(* CODESYS project string-builder-unit-test-history

Project tree, tasks and I/O mapping:
  Device : CODESYS Control Win V3 x64, 3S - Smart Software Solutions GmbH, version 3.5.17.20
    application Application
      libraries: Standard, 3.5.18.0 (System); co♻e - A unittest framework for CODESYS, 1.2.0.0 (www.co5e.org); StringBuilder, 0.0.0.1 (PowerCore Engineering)
      task MainTask (cyclic, interval t#20ms, priority 1) calls PLC_PRG
      function block FB_TestSuite_withBuffer [ST]: AssertEquals_Buffer
      FunctionBlocks/
        function block UT_StringBuilder [ST]: T001_Append, T002_Reset
        function block UT_StringBuilderExt [ST]: T001_Append, T002_Reset
      Functions/
        function block UT_ANY_TO_HEXSTR [ST]: T001_Test
        function block UT_ANY_TO_NUMSTRING [ST]: T001_Test
        function block UT_FindFormat [ST]: T001_FindFormat
        function block UT_Format_1 [ST]: T001_Format_1
        function block UT_Format [ST]: T001_Format_2, T002_Format_3, T003_Format_4, T004_Format_5, T005_Format_6, T006_Format_7, T007_Format_8, T008_Format_9, T009_Format_10, T010_Format_2
        function block UT_FormatExt_1 [ST]: T001_Format_1
        function block UT_FormatExt [ST]: T001_FormatExt_2, T002_FormatExt_3, T003_FormatExt_4, T004_FormatExt_5, T005_FormatExt_6, T006_FormatExt_7, T007_FormatExt_8, T008_FormatExt_9, T009_FormatExt_10, T010_FormatExt_2
      program PLC_PRG [ST]
*)

// Device/Application/PLC_PRG
PROGRAM PLC_PRG
VAR
	utStringBuilder : UT_StringBuilder;
	utFindFormat : UT_FindFormat;
	utFormat_1 : UT_Format_1;
	utFormat : UT_Format;
END_VAR

coUnit.RUN();

END_PROGRAM

// Device/Application/FunctionBlocks/UT_StringBuilder
FUNCTION_BLOCK UT_StringBuilder EXTENDS coUnit.FB_TestSuite
VAR_INPUT
END_VAR
VAR_OUTPUT
END_VAR
VAR
END_VAR

T001_Append();
T002_Reset();

METHOD T001_Append
VAR_INPUT
END_VAR
VAR
	sb : PSB.StringBuilder;
END_VAR
TEST('T001_Append');

sb.Append('Hello');
sb.Append(', ');
sb.Append('world!');

AssertEquals_STRING('Hello, world!', sb.sOutput, 'Unexpected result');

TEST_FINISHED();
END_METHOD

METHOD T002_Reset
VAR_INPUT
END_VAR
VAR
	sb : PSB.StringBuilder;
END_VAR
TEST('T002_Reset');

sb.Append('Hello, world!');

AssertEquals_STRING('Hello, world!', sb.sOutput, 'Unexpected result');

sb.Reset();
AssertEquals_STRING('', sb.sOutput, 'Unexpected result');

TEST_FINISHED();
END_METHOD

END_FUNCTION_BLOCK

// Device/Application/Functions/UT_FindFormat
FUNCTION_BLOCK UT_FindFormat EXTENDS coUnit.FB_TestSuite
VAR_INPUT
END_VAR
VAR_OUTPUT
END_VAR
VAR
END_VAR

T001_FindFormat('This {} thing', start:=0, sl_start:=6, sl_end:=7);
T001_FindFormat('{} thing', start:=0, sl_start:=1, sl_end:=2);
T001_FindFormat('thing', start:=0, sl_start:=0, sl_end:=0);
T001_FindFormat('This {} thing {}', start:=7, sl_start:=15, sl_end:=16);

METHOD T001_FindFormat
VAR_INPUT
	sFmtStr : STRING(255);
	start : DINT;
	sl_start : DINT;
	sl_end : DINT;
END_VAR
VAR
	slResult : PSB.slice;
END_VAR
TEST(concat(concat('T001_FindFormat:', sFmtStr), concat(concat('-', DINT_TO_STRING(start)), 
	concat(concat('-' , TO_STRING(sl_start)), concat('-', TO_STRING(sl_end)))))); 

slResult := PSB.FindFormat(sFmtStr, start);

AssertEquals_DINT(sl_start, slResult.start, 'Unexpected start position');
AssertEquals_DINT(sl_end, slResult.end, 'Unexpected end position');

TEST_FINISHED();
END_METHOD

END_FUNCTION_BLOCK

// Device/Application/Functions/UT_Format_1
FUNCTION_BLOCK UT_Format_1 EXTENDS coUnit.FB_TestSuite
VAR_INPUT
END_VAR
VAR_OUTPUT
END_VAR
VAR
END_VAR

T001_Format_1('Hello, {}!', 'world', 'Hello, world!');
T001_Format_1('Hello {}', 'john', 'Hello john');

METHOD T001_Format_1
VAR_INPUT
	fmtstr : STRING(255);
	str1 : STRING(255);
	sExpected : STRING(255);
END_VAR
VAR
	sResult : STRING(255);
END_VAR
TEST(concat(concat('T001_Format_1:', fmtstr), concat('-', str1)));

sResult := PSB.Format_1(fmtstr, str1);

AssertEquals_STRING(sExpected, sResult, 'unexpected result');

TEST_FINISHED();
END_METHOD

END_FUNCTION_BLOCK

// Device/Application/Functions/UT_Format
FUNCTION_BLOCK UT_Format EXTENDS coUnit.FB_TestSuite
VAR_INPUT
END_VAR
VAR_OUTPUT
END_VAR
VAR
END_VAR

T001_Format_2('Hello, {}! Goodbye {} world.',
              'world',
              'cruel',
              'Hello, world! Goodbye cruel world.');
T002_Format_3('{}-{}-{}',
	'a',
	'b',
	'c',
	'a-b-c');
T003_Format_4('{}-{}-{}-{}-',
	'1',
	'2',
	'3',
	'4',
	'1-2-3-4-');
// missing format element
T004_Format_5('{}-{}-{}-{}-',
	'1',
	'2',
	'3',
	'4',
	'5',
	'1-2-3-4-');
	
// extra format element
T004_Format_5('{}-{}-{}-{}-{}-{}',
	'1',
	'2',
	'3',
	'4',
	'5',
	'1-2-3-4-5-{}');
T005_Format_6('{}-{}-{}-{}-{}-{}',
	INT_TO_STRING(1),
	TO_STRING(123.456),
	'c',
	'd',
	'e',
	'f',
	'1-123.456-c-d-e-f');
T006_Format_7('{}-{}-{}-{}-{}-{}-{}',
	'1', '2', '3', '4', '5', '6', '7',
	'1-2-3-4-5-6-7');
T007_Format_8('{}-{}-{}-{}-{}-{}-{}-{}',
	'1', '2', '3', '4', '5', '6', '7','8',
	'1-2-3-4-5-6-7-8');
T008_Format_9('{}-{}-{}-{}-{}-{}-{}-{}-{}',
	'1', '2', '3', '4', '5', '6', '7','8','9',
	'1-2-3-4-5-6-7-8-9');
T009_Format_10('{}-{}-{}-{}-{}-{}-{}-{}-{}-{}',
	'1', '2', '3', '4', '5', '6', '7','8','9','10',
	'1-2-3-4-5-6-7-8-9-10');
T010_Format_2('test-with-to-string-input-int:{}-real:{}', 123, 456.789, 'test-with-to-string-input-int:123-real:456.789');

METHOD T001_Format_2
VAR_INPUT
	fmtstr : STRING(255);
	str1 : STRING(255);
	str2 : STRING(255);
	sExpected : STRING(255);
END_VAR
VAR_INST
	sResult : STRING(255);
END_VAR
TEST(concat(concat('T001_Format_2:', fmtstr), concat('-', sExpected)));

sResult := PSB.Format_2(fmtstr, str1, str2);

AssertEquals_STRING(sExpected, sResult, 'unexpected result');

TEST_FINISHED();
END_METHOD

METHOD T002_Format_3
VAR_INPUT
	fmtstr : STRING(255);
	str1 : STRING(255);
	str2 : STRING(255);
	str3 : STRING(255);
	sExpected : STRING(255);
END_VAR
VAR_INST
	sResult : STRING(255);
END_VAR
TEST(concat(concat('T001_Format_3:', fmtstr), concat('-', sExpected)));

sResult := PSB.Format_3(fmtstr, str1, str2, str3);

AssertEquals_STRING(sExpected, sResult, 'unexpected result');

TEST_FINISHED();
END_METHOD

METHOD T003_Format_4
VAR_INPUT
	fmtstr : STRING(255);
	str1 : STRING(255);
	str2 : STRING(255);
	str3 : STRING(255);
	str4 : STRING(255);
	sExpected : STRING(255);
END_VAR
VAR_INST
	sResult : STRING(255);
END_VAR
TEST(concat(concat('T003_Format_4:', fmtstr), concat('-', sExpected)));

sResult := PSB.Format_4(fmtstr, str1, str2, str3, str4);

AssertEquals_STRING(sExpected, sResult, 'unexpected result');

TEST_FINISHED();
END_METHOD

METHOD T004_Format_5
VAR_INPUT
	fmtstr : STRING(255);
	str1 : STRING(255);
	str2 : STRING(255);
	str3 : STRING(255);
	str4 : STRING(255);
	str5 : STRING(255);
	sExpected : STRING(255);
END_VAR
VAR_INST
	sResult : STRING(255);
END_VAR
TEST(concat(concat('T004_Format_5:', fmtstr), concat('-', sExpected)));

sResult := PSB.Format_5(fmtstr, str1, str2, str3, str4, str5);

AssertEquals_STRING(sExpected, sResult, 'unexpected result');

TEST_FINISHED();
END_METHOD

METHOD T005_Format_6
VAR_INPUT
	fmtstr : STRING(255);
	str1 : STRING(255);
	str2 : STRING(255);
	str3 : STRING(255);
	str4 : STRING(255);
	str5 : STRING(255);
	str6 : STRING(255);
	sExpected : STRING(255);
END_VAR
VAR_INST
	sResult : STRING(255);
END_VAR
TEST(concat(concat('T005_Format_6:', fmtstr), concat('-', sExpected)));

sResult := PSB.Format_6(fmtstr, str1, str2, str3, str4, str5, str6);

AssertEquals_STRING(sExpected, sResult, 'unexpected result');

TEST_FINISHED();
END_METHOD

METHOD T006_Format_7
VAR_INPUT
	fmtstr : STRING(255);
	str1 : STRING(255);
	str2 : STRING(255);
	str3 : STRING(255);
	str4 : STRING(255);
	str5 : STRING(255);
	str6 : STRING(255);
	str7 : STRING(255);
	sExpected : STRING(255);
END_VAR
VAR_INST
	sResult : STRING(255);
END_VAR
TEST(concat(concat('T006_Format_7:', fmtstr), concat('-', sExpected)));

sResult := PSB.Format_7(fmtstr, str1, str2, str3, str4, str5, str6, str7);

AssertEquals_STRING(sExpected, sResult, 'unexpected result');

TEST_FINISHED();
END_METHOD

METHOD T007_Format_8
VAR_INPUT
	fmtstr : STRING(255);
	str1 : STRING(255);
	str2 : STRING(255);
	str3 : STRING(255);
	str4 : STRING(255);
	str5 : STRING(255);
	str6 : STRING(255);
	str7 : STRING(255);
	str8 : STRING(255);
	sExpected : STRING(255);
END_VAR
VAR_INST
	sResult : STRING(255);
END_VAR
TEST(concat(concat('T007_Format_8:', fmtstr), concat('-', sExpected)));

sResult := PSB.Format_8(fmtstr, str1, str2, str3, str4, str5, str6, str7, str8);

AssertEquals_STRING(sExpected, sResult, 'unexpected result');

TEST_FINISHED();
END_METHOD

METHOD T008_Format_9
VAR_INPUT
	fmtstr : STRING(255);
	str1 : STRING(255);
	str2 : STRING(255);
	str3 : STRING(255);
	str4 : STRING(255);
	str5 : STRING(255);
	str6 : STRING(255);
	str7 : STRING(255);
	str8 : STRING(255);
	str9 : STRING(255);
	sExpected : STRING(255);
END_VAR
VAR_INST
	sResult : STRING(255);
END_VAR
TEST(concat(concat('T008_Format_9:', fmtstr), concat('-', sExpected)));

sResult := PSB.Format_9(fmtstr, str1, str2, str3, str4, str5, str6, str7, str8, str9);

AssertEquals_STRING(sExpected, sResult, 'unexpected result');

TEST_FINISHED();
END_METHOD

METHOD T009_Format_10
VAR_INPUT
	fmtstr : STRING(255);
	str1 : STRING(255);
	str2 : STRING(255);
	str3 : STRING(255);
	str4 : STRING(255);
	str5 : STRING(255);
	str6 : STRING(255);
	str7 : STRING(255);
	str8 : STRING(255);
	str9 : STRING(255);
	str10 : STRING(255);
	sExpected : STRING(255);
END_VAR
VAR_INST
	sResult : STRING(255);
END_VAR
TEST(concat(concat('T009_Format_10:', fmtstr), concat('-', sExpected)));

sResult := PSB.Format_10(fmtstr, str1, str2, str3, str4, str5, str6, str7, str8, str9, str10);

AssertEquals_STRING(sExpected, sResult, 'unexpected result');

TEST_FINISHED();
END_METHOD

METHOD T010_Format_2
VAR_INPUT
	fmtstr : STRING(255);
	i : INT;
	rl : REAL;
	sExpected : STRING(255);
END_VAR
VAR_INST
	sResult : STRING(255);
END_VAR
TEST(concat(concat('T010_Format_2:', fmtstr), concat('-', sExpected)));

sResult := PSB.Format_2(fmtstr, TO_STRING(i), TO_STRING(rl));

AssertEquals_STRING(sExpected, sResult, 'unexpected result');

TEST_FINISHED();
END_METHOD

END_FUNCTION_BLOCK

// Device/Application/FB_TestSuite_withBuffer
FUNCTION_BLOCK FB_TestSuite_withBuffer EXTENDS coUnit.FB_TestSuite
VAR_INPUT
END_VAR
VAR_OUTPUT
END_VAR
VAR
END_VAR

METHOD AssertEquals_Buffer
VAR_INPUT
	// Expected
	pe : POINTER TO ARRAY [0..32767] OF BYTE;
	// Actual
	pa : POINTER TO ARRAY [0..32767] OF BYTE;
	// Size
	sz : UINT;
END_VAR
VAR
	ix : UINT;
	xDifferent : BOOL;
END_VAR
FOR ix := 0 TO sz BY 1 DO
	IF pa^[ix] <> 0 AND pe^[ix] <> 0 THEN
		IF pa^[ix] <> pe^[ix] THEN
			xDifferent := TRUE;
			EXIT;
		END_IF
	ELSIF pa^[ix] = 0 AND pe^[ix] = 0 THEN
		EXIT;
	ELSE
		xDifferent := TRUE;
		EXIT;
	END_IF
END_FOR

AssertFalse(xDifferent, concat('Buffers found to differ at index: ', UINT_TO_STRING(ix)));
END_METHOD

END_FUNCTION_BLOCK

// Device/Application/FunctionBlocks/UT_StringBuilderExt
FUNCTION_BLOCK UT_StringBuilderExt EXTENDS FB_TestSuite_withBuffer
VAR_INPUT
END_VAR
VAR_OUTPUT
END_VAR
VAR
END_VAR

T001_Append();
T002_Reset();

METHOD T001_Append
VAR_INPUT
END_VAR
VAR
	sExpected : STRING(512) := 'wwwwwwwwwwwwwwwwwwwwwwwwwwwwwwwwwwwwwwwwwwwwwwwwwwwwwwwwwwwwwwwwwwwwwwwwwwwwwwwwwwwwwwwwwwwwwwwwwwwwwwwwwwwwwwwwwwwwwwwwwwwwwwwwxxxxxxxxxxxxxxxxxxxxxxxxxxxxxxxxxxxxxxxxxxxxxxxxxxxxxxxxxxxxxxxxxxxxxxxxxxxxxxxxxxxxxxxxxxxxxxxxxxxxxxxxxxxxxxxxxxxxxxxxxxxxxxxxyyyyyyyyyyyyyyyyyyyyyyyyyyyyyyyyyyyyyyyyyyyyyyyyyyyyyyyyyyyyyyyyyyyyyyyyyyyyyyyyyyyyyyyyyyyyyyyyyyyyyyyyyyyyyyyyyyyyyyyyyyyyyyyyzzzzzzzzzzzzzzzzzzzzzzzzzzzzzzzzzzzzzzzzzzzzzzzzzzzzzzzzzzzzzzzzzzzzzzzzzzzzzzzzzzzzzzzzzzzzzzzzzzzzzzzzzzzzzzzzzzzzzzzzzzzzzzzz';
	sBuffer : STRING(512);
	sb : PSB.StringBuilderExt := (pBuffer:=ADR(sBuffer), szBuffer:=SIZEOF(sBuffer));
END_VAR
TEST('T001_Append');

sb.Append('wwwwwwwwwwwwwwwwwwwwwwwwwwwwwwwwwwwwwwwwwwwwwwwwwwwwwwwwwwwwwwwwwwwwwwwwwwwwwwwwwwwwwwwwwwwwwwwwwwwwwwwwwwwwwwwwwwwwwwwwwwwwwwww');
sb.Append('xxxxxxxxxxxxxxxxxxxxxxxxxxxxxxxxxxxxxxxxxxxxxxxxxxxxxxxxxxxxxxxxxxxxxxxxxxxxxxxxxxxxxxxxxxxxxxxxxxxxxxxxxxxxxxxxxxxxxxxxxxxxxxxx');
sb.Append('yyyyyyyyyyyyyyyyyyyyyyyyyyyyyyyyyyyyyyyyyyyyyyyyyyyyyyyyyyyyyyyyyyyyyyyyyyyyyyyyyyyyyyyyyyyyyyyyyyyyyyyyyyyyyyyyyyyyyyyyyyyyyyyy');
sb.Append('zzzzzzzzzzzzzzzzzzzzzzzzzzzzzzzzzzzzzzzzzzzzzzzzzzzzzzzzzzzzzzzzzzzzzzzzzzzzzzzzzzzzzzzzzzzzzzzzzzzzzzzzzzzzzzzzzzzzzzzzzzzzzzzz');
sb.Append('this wont append');

AssertEquals_Buffer(ADR(sBuffer), ADR(sExpected), SIZEOF(sBuffer));

TEST_FINISHED();
END_METHOD

METHOD T002_Reset
VAR_INPUT
END_VAR
VAR
	sBuffer : STRING(512);
	sb : PSB.StringBuilderExt := (pBuffer:=ADR(sBuffer), szBuffer:=SIZEOF(sBuffer));
END_VAR
TEST('T002_Reset');

sb.Append('Hello, world!');

AssertEquals_STRING('Hello, world!', sBuffer, 'Unexpected result');

sb.Reset();
AssertEquals_STRING('', sBuffer, 'Unexpected result');

TEST_FINISHED();
END_METHOD

END_FUNCTION_BLOCK

// Device/Application/Functions/UT_ANY_TO_HEXSTR
FUNCTION_BLOCK UT_ANY_TO_HEXSTR EXTENDS coUnit.FB_TestSuite
VAR_INPUT
END_VAR
VAR_OUTPUT
END_VAR
VAR
	xw : __XWORD := 16#DEADBEEF;
	w : WORD := 16#BEEF;
	str : STRING := 'a';
	i : INT := -1;
	pstr : POINTER TO BYTE;
	pxw : __XWORD;
END_VAR

T001_Test('__xword-lo-case-64bit-pad',
		sResult:=PSB.ANY_TO_HEXSTR(xw, 16, TRUE),
		sExpected:='00000000deadbeef'
);
T001_Test('word-up-case-16bit-pad',
		sResult:=PSB.ANY_TO_HEXSTR(w, 4, FALSE),
		sExpected:='BEEF'
);
pstr := ADR(str);
pxw := pstr;
T001_Test('str-lo-case-0bit-pad',
		sResult:=PSB.ANY_TO_HEXSTR(str, 0, TRUE),
		sExpected:=PSB.ANY_TO_HEXSTR(pxw, 4, TRUE)
);
T001_Test('int-lo-case-16bit-pad',
		sResult:=PSB.ANY_TO_HEXSTR(i, 4, TRUE),
		sExpected:='ffffffff' // in Codesys Win V3 x64 INT is actually represented with 32bit value
);

METHOD T001_Test
VAR_INPUT
	sTestName : STRING(255);
	sResult : STRING(255);
	sExpected : STRING(255);
END_VAR
TEST(sTestName);

AssertEquals_STRING(sExpected, sResult, 'Unexpected result');

TEST_FINISHED();
END_METHOD

END_FUNCTION_BLOCK

// Device/Application/Functions/UT_ANY_TO_NUMSTRING
FUNCTION_BLOCK UT_ANY_TO_NUMSTRING EXTENDS coUnit.FB_TestSuite
VAR_INPUT
END_VAR
VAR_OUTPUT
END_VAR
VAR
	xw : __XWORD := 16#DEADBEEF;
	w : WORD := 16#BEEF;
	str : STRING := 'a';
	i : INT := -1;
	pstr : POINTER TO BYTE;
	pxw : __XWORD;
	options : PSB.FormatOptions := (sFill:='0', align:=PSB.Alignment.Right);
	
	_BOOL : BOOL;
	//_BIT : BIT; // TODO: make a struct with bits and pass it
	_BYTE : BYTE;
	_WORD : WORD;
	_DWORD : DWORD;
	_LWORD : LWORD;
	_SINT : SINT;
	_INT : INT;
	_DINT : DINT;
	_LINT : LINT;
	_USINT : USINT;
	_UINT : UINT;
	_UDINT : UDINT;
	_ULINT : ULINT;
	_REAL : REAL;
	_LREAL : LREAL;
	_STRING : STRING;
	_WSTRING : WSTRING;
	_TIME : TIME;
	_DATE : DATE;
	_DATEANDTIME : DT;
	_TIMEOFDAY : TOD;
	_POINTER : POINTER TO BYTE;
	_REFERENCE : REFERENCE TO BYTE;
	_LTIME : LTIME;
	_LDATE : LDATE;
	_LDT : LDT;

END_VAR

options.iMinWidth := 16;
T001_Test('__xword-lo-case-64bit-pad',
		sResult:=PSB.ANY_TO_NUMSTRING(xw, 16, TRUE, options),
		sExpected:='00000000deadbeef'
);
options.iMinWidth := 4;
T001_Test('word-up-case-16bit-pad',
		sResult:=PSB.ANY_TO_NUMSTRING(w, 16, FALSE, options),
		sExpected:='BEEF'
);
pstr := ADR(str);
pxw := pstr;
options.iMinWidth := -1;
T001_Test('str-lo-case-0bit-pad',
		sResult:=PSB.ANY_TO_NUMSTRING(str, 16, TRUE, options),
		sExpected:=PSB.ANY_TO_NUMSTRING(pxw, 16, TRUE, options)
);
options.iMinWidth := 4;
T001_Test('neg-int-lo-case-16bit-pad',
		sResult:=PSB.ANY_TO_NUMSTRING(i, 16, TRUE, options),
		sExpected:='00-1'
);
w := INT_TO_WORD(i);
T001_Test('neg-int-to-word-lo-case-16bit-pad',
		sResult:=PSB.ANY_TO_NUMSTRING(w, 16, TRUE, options),
		sExpected:='ffff'
);

options.iMinWidth := -1;
_BOOL := TRUE;
T001_Test('_BOOL-lo-case-no-pad',
	sResult:=PSB.ANY_TO_NUMSTRING(_BOOL, 16, TRUE, options),
	sExpected:='1'
);

// _BIT := 1;
// T001_Test('_BIT-lo-case-no-pad',
// 	sResult:=PSB.ANY_TO_NUMSTRING(_BIT, 16, TRUE, options),
// 	sExpected:=''
// );

_BYTE := 123;
T001_Test('_BYTE-lo-case-no-pad',
	sResult:=PSB.ANY_TO_NUMSTRING(_BYTE, 16, TRUE, options),
	sExpected:='7b'
);

_WORD := 16#1234;
T001_Test('_WORD-lo-case-no-pad',
	sResult:=PSB.ANY_TO_NUMSTRING(_WORD, 16, TRUE, options),
	sExpected:='1234'
);

_DWORD := INT_TO_DWORD(-2);
T001_Test('_DWORD-lo-case-no-pad',
	sResult:=PSB.ANY_TO_NUMSTRING(_DWORD, 16, TRUE, options),
	sExpected:='fffffffe'
);

_LWORD := 16#F234_4321_ABCD_EF12;
T001_Test('_LWORD-lo-case-no-pad',
	sResult:=PSB.ANY_TO_NUMSTRING(_LWORD, 16, TRUE, options),
	sExpected:='f2344321abcdef12'
);

_SINT := 1;
T001_Test('_SINT-lo-case-no-pad',
	sResult:=PSB.ANY_TO_NUMSTRING(_SINT, 16, TRUE, options),
	sExpected:='1'
);

_INT := 1000;
T001_Test('_INT-lo-case-no-pad',
	sResult:=PSB.ANY_TO_NUMSTRING(_INT, 16, TRUE, options),
	sExpected:='3e8'
);

_DINT := 20000;
T001_Test('_DINT-lo-case-no-pad',
	sResult:=PSB.ANY_TO_NUMSTRING(_DINT, 16, TRUE, options),
	sExpected:='4e20'
);

_LINT := 9223372036854775807;
T001_Test('_LINT-lo-case-no-pad',
	sResult:=PSB.ANY_TO_NUMSTRING(_LINT, 16, TRUE, options),
	sExpected:='7fffffffffffffff'
);

_USINT := 10;
T001_Test('_USINT-lo-case-no-pad',
	sResult:=PSB.ANY_TO_NUMSTRING(_USINT, 16, TRUE, options),
	sExpected:='a'
);

_UINT := 16#FFFF;
T001_Test('_UINT-lo-case-no-pad',
	sResult:=PSB.ANY_TO_NUMSTRING(_UINT, 16, TRUE, options),
	sExpected:='ffff'
);

_UDINT := 16#DEADBEEF;
T001_Test('_UDINT-lo-case-no-pad',
	sResult:=PSB.ANY_TO_NUMSTRING(_UDINT, 16, TRUE, options),
	sExpected:='deadbeef'
);

_ULINT := 16#DEADDEADBEEF;
T001_Test('_ULINT-lo-case-no-pad',
	sResult:=PSB.ANY_TO_NUMSTRING(_ULINT, 16, TRUE, options),
	sExpected:='deaddeadbeef'
);

_REAL := 1;
T001_Test('_REAL-lo-case-no-pad',
	sResult:=PSB.ANY_TO_NUMSTRING(_REAL, 16, TRUE, options),
	sExpected:='3f800000'
);

_LREAL := 1;
T001_Test('_LREAL-lo-case-no-pad',
	sResult:=PSB.ANY_TO_NUMSTRING(_LREAL, 16, TRUE, options),
	sExpected:='3ff0000000000000'
);

_STRING := ' ';
pxw := ADR(_STRING);
T001_Test('_STRING-lo-case-no-pad',
	sResult:=PSB.ANY_TO_NUMSTRING(_STRING, 16, TRUE, options),
	sExpected:=PSB.ANY_TO_NUMSTRING(pxw, 16, TRUE, options)
);

_WSTRING := " ";
pxw := ADR(_WSTRING);
T001_Test('_WSTRING-lo-case-no-pad',
	sResult:=PSB.ANY_TO_NUMSTRING(_WSTRING, 16, TRUE, options),
	sExpected:=PSB.ANY_TO_NUMSTRING(pxw, 16, TRUE, options)
);

_TIME := T#1S;
T001_Test('_TIME-lo-case-no-pad',
	sResult:=PSB.ANY_TO_NUMSTRING(_TIME, 16, TRUE, options),
	sExpected:='3e8'
);

_DATE := DATE#2022-6-2;
T001_Test('_DATE-lo-case-no-pad',
	sResult:=PSB.ANY_TO_NUMSTRING(_DATE, 16, TRUE, options),
	sExpected:='6297fd80'
);

_DATEANDTIME := DT#2022-6-2-15:10:00;
T001_Test('_DATEANDTIME-lo-case-no-pad',
	sResult:=PSB.ANY_TO_NUMSTRING(_DATEANDTIME, 16, TRUE, options),
	sExpected:='6298d2c8'
);

_TIMEOFDAY := TOD#15:10:00;
T001_Test('_TIMEOFDAY-lo-case-no-pad',
	sResult:=PSB.ANY_TO_NUMSTRING(_TIMEOFDAY, 16, TRUE, options),
	sExpected:='3412140'
);

_POINTER := ADR(_BYTE);
pxw := ADR(_POINTER);
T001_Test('_POINTER-lo-case-no-pad',
	sResult:=PSB.ANY_TO_NUMSTRING(_POINTER, 16, TRUE, options),
	sExpected:=PSB.ANY_TO_NUMSTRING(pxw, 16, TRUE, options)
);

_REFERENCE REF=_BYTE;
pxw := ADR(_BYTE);
T001_Test('_REFERENCE-lo-case-no-pad',
	sResult:=PSB.ANY_TO_NUMSTRING(_REFERENCE, 16, TRUE, options),
	sExpected:=PSB.ANY_TO_NUMSTRING(pxw, 16, TRUE, options)
);

_LTIME := LTIME#1S;
T001_Test('_LTIME-lo-case-no-pad',
	sResult:=PSB.ANY_TO_NUMSTRING(_LTIME, 16, TRUE, options),
	sExpected:='3b9aca00'
);

_LDATE := LDATE#2022-6-2;
T001_Test('_LDATE-lo-case-no-pad',
	sResult:=PSB.ANY_TO_NUMSTRING(_LDATE, 16, TRUE, options),
	sExpected:='16f4a4a6ed070000'
);

_LDT := LDT#2022-6-2-15:29:00;
T001_Test('_LDT-lo-case-no-pad',
	sResult:=PSB.ANY_TO_NUMSTRING(_LDT, 16, TRUE, options),
	sExpected:='16f4d758e7ed5800'
);

_WORD := 8#644;
T001_Test('_WORD-lo-case-no-pad-oct',
	sResult:=PSB.ANY_TO_NUMSTRING(_WORD, 8, TRUE, options),
	sExpected:='644'
);

_BYTE := 2#1010_0101;
T001_Test('_BYTE-lo-case-no-pad-bin',
	sResult:=PSB.ANY_TO_NUMSTRING(_BYTE, 2, TRUE, options),
	sExpected:='10100101'
);

METHOD T001_Test
VAR_INPUT
	sTestName : STRING(255);
	sResult : STRING(255);
	sExpected : STRING(255);
END_VAR
VAR
	pa : POINTER TO ARRAY [0..3200] OF BYTE;
END_VAR
pa := ADR(sTestName) - 100;

TEST(sTestName);

AssertEquals_STRING(sExpected, sResult, 'Unexpected result');

TEST_FINISHED();
END_METHOD

END_FUNCTION_BLOCK

// Device/Application/Functions/UT_FormatExt_1
FUNCTION_BLOCK UT_FormatExt_1 EXTENDS FB_TestSuite_withBuffer
VAR_INPUT
END_VAR
VAR_OUTPUT
END_VAR
VAR
END_VAR

T001_Format_1('Hello, {}!', 'world', 'Hello, world!');
T001_Format_1('Hello {}', 'john', 'Hello john');
// Should truncate
T001_Format_1('zz{}zzzzzzzzzzzzzzzzzzzzzzzzzzzzzzzzzzzzzzzzzzzzzzzzzzzzzzzzzzzzzzzzzzzzzzzzzzzzzzzzzzzzzzzzzzzzzzzzzzzzzzzzzzzzzzzzzzzzzzzzzzzzzzzzzzzzzzzzzzzzzzzzzzzzzzzzzzzzzzzzzzzzzzzzzzzzzzzzzzzzzzzzzzzzzzzzzzzzzzzzzzzzzzzzzzzzzzzzzzzzzzzzzzzzzzzzzzzzzzzzzzzzzzzzzzz',
	'XXXXXXXXXXXXXXXXXXXXXXXXXXXXXXXXXXXXXXXXXXXXXXXXXXXXXXXXXXXXXXXXXXXXXXXXXXXXXXXXXXXXXXXXXXXXXXXXXXXXXXXXXXXXXXXXXXXXXXXXXXXXXXXXXXXXXXXXXXXXXXXXXXXXXXXXXXXXXXXXXXXXXXXXXXXXXXXXXXXXXXXXXXXXXXXXXXXXXXXXXXXXXXXXXXXXXXXXXXXXXXXXXXXXXXXXXXXXXXXXXXXXXXXXXXXXXXX',
	'zzXXXXXXXXXXXXXXXXXXXXXXXXXXXXXXXXXXXXXXXXXXXXXXXXXXXXXXXXXXXXXXXXXXXXXXXXXXXXXXXXXXXXXXXXXXXXXXXXXXXXXXXXXXXXXXXXXXXXXXXXXXXXXXXXXXXXXXXXXXXXXXXXXXXXXXXXXXXXXXXXXXXXXXXXXXXXXXXXXXXXXXXXXXXXXXXXXXXXXXXXXXXXXXXXXXXXXXXXXXXXXXXXXXXXXXXXXXXXXXXXXXXXXXXXXXXXXXXzzzzzzzzzzzzzzzzzzzzzzzzzzzzzzzzzzzzzzzzzzzzzzzzzzzzzzzzzzzzzzzzzzzzzzzzzzzzzzzzzzzzzzzzzzzzzzzzzzzzzzzzzzzzzzzzzzzzzzzzzzzzzzzzzzzzzzzzzzzzzzzzzzzzzzzzzzzzzzzzzzzzzzzzzzzzzzzzzzzzzzzzzzzzzzzzzzzzzzzzzzzzzzzzzzzzzzzzzzzzzzzzzzzzzzzzzzzzzzzzzzz'
);

METHOD T001_Format_1
VAR_INPUT
	fmtstr : STRING(255);
	str1 : STRING(255);
	sExpected : STRING(500);
END_VAR
VAR
	sResult : STRING(500);
	sb : PSB.StringBuilderExt := (pBuffer:=ADR(sResult), szBuffer:=SIZEOF(sResult));
END_VAR
TEST(concat(concat('T001_Format_1:', fmtstr), concat('-', str1)));

PSB.FormatExt_1(sb, fmtstr, str1);

AssertEquals_Buffer(ADR(sExpected), ADR(sResult), SIZEOF(sResult));

TEST_FINISHED();
END_METHOD

END_FUNCTION_BLOCK

// Device/Application/Functions/UT_FormatExt
FUNCTION_BLOCK UT_FormatExt EXTENDS FB_TestSuite_withBuffer
VAR_INPUT
END_VAR
VAR_OUTPUT
END_VAR
VAR
END_VAR

T001_FormatExt_2('Hello, {}! Goodbye {} world.',
              'world',
              'cruel',
              'Hello, world! Goodbye cruel world.');
T002_FormatExt_3('{}-{}-{}',
	'a',
	'b',
	'c',
	'a-b-c');
T003_FormatExt_4('{}-{}-{}-{}-',
	'1',
	'2',
	'3',
	'4',
	'1-2-3-4-');
// missing format element
T004_FormatExt_5('{}-{}-{}-{}-',
	'1',
	'2',
	'3',
	'4',
	'5',
	'1-2-3-4-');
	
// extra format element
T004_FormatExt_5('{}-{}-{}-{}-{}-{}',
	'1',
	'2',
	'3',
	'4',
	'5',
	'1-2-3-4-5-{}');
T005_FormatExt_6('{}-{}-{}-{}-{}-{}',
	INT_TO_STRING(1),
	TO_STRING(123.456),
	'c',
	'd',
	'e',
	'f',
	'1-123.456-c-d-e-f');
T006_FormatExt_7('{}-{}-{}-{}-{}-{}-{}',
	'1', '2', '3', '4', '5', '6', '7',
	'1-2-3-4-5-6-7');
T007_FormatExt_8('{}-{}-{}-{}-{}-{}-{}-{}',
	'1', '2', '3', '4', '5', '6', '7','8',
	'1-2-3-4-5-6-7-8');
T008_FormatExt_9('{}-{}-{}-{}-{}-{}-{}-{}-{}',
	'1', '2', '3', '4', '5', '6', '7','8','9',
	'1-2-3-4-5-6-7-8-9');
T009_FormatExt_10('{}-{}-{}-{}-{}-{}-{}-{}-{}-{}',
	'1', '2', '3', '4', '5', '6', '7','8','9','10',
	'1-2-3-4-5-6-7-8-9-10');
T010_FormatExt_2('test-with-to-string-input-int:{}-real:{}', 123, 456.789, 'test-with-to-string-input-int:123-real:456.789');

METHOD T001_FormatExt_2
VAR_INPUT
	fmtstr : STRING(255);
	str1 : STRING(255);
	str2 : STRING(255);
	sExpected : STRING(500);
END_VAR
VAR_INST
	sResult : STRING(500);
	sb : PSB.StringBuilderExt;
END_VAR
TEST(concat(concat('T001_Format_2:', fmtstr), concat('-', sExpected)));

sb.pBuffer := ADR(sResult);
sb.szBuffer := SIZEOF(sResult);

PSB.FormatExt_2(sb, fmtstr, str1, str2);

AssertEquals_Buffer(ADR(sExpected), ADR(sResult), SIZEOF(sResult));
sb.Reset();
TEST_FINISHED();
END_METHOD

METHOD T002_FormatExt_3
VAR_INPUT
	fmtstr : STRING(255);
	str1 : STRING(255);
	str2 : STRING(255);
	str3 : STRING(255);
	sExpected : STRING(500);
END_VAR
VAR_INST
	sResult : STRING(500);
	sb : PSB.StringBuilderExt;
END_VAR
TEST(concat(concat('T001_Format_3:', fmtstr), concat('-', sExpected)));

sb.pBuffer := ADR(sResult);
sb.szBuffer := SIZEOF(sResult);

PSB.FormatExt_3(sb, fmtstr, str1, str2, str3);

AssertEquals_Buffer(ADR(sExpected), ADR(sResult), sizeof(sResult));
sb.Reset();
TEST_FINISHED();
END_METHOD

METHOD T003_FormatExt_4
VAR_INPUT
	fmtstr : STRING(255);
	str1 : STRING(255);
	str2 : STRING(255);
	str3 : STRING(255);
	str4 : STRING(255);
	sExpected : STRING(500);
END_VAR
VAR_INST
	sResult : STRING(500);
	sb : PSB.StringBuilderExt;
END_VAR
TEST(concat(concat('T003_Format_4:', fmtstr), concat('-', sExpected)));

sb.pBuffer := ADR(sResult);
sb.szBuffer := SIZEOF(sResult);

PSB.FormatExt_4(sb, fmtstr, str1, str2, str3, str4);

AssertEquals_Buffer(ADR(sExpected), ADR(sResult), sizeof(sResult));
sb.Reset();
TEST_FINISHED();
END_METHOD

METHOD T004_FormatExt_5
VAR_INPUT
	fmtstr : STRING(255);
	str1 : STRING(255);
	str2 : STRING(255);
	str3 : STRING(255);
	str4 : STRING(255);
	str5 : STRING(255);
	sExpected : STRING(500);
END_VAR
VAR_INST
	sResult : STRING(500);
	sb : PSB.StringBuilderExt;
END_VAR
TEST(concat(concat('T004_Format_5:', fmtstr), concat('-', sExpected)));

sb.pBuffer := ADR(sResult);
sb.szBuffer := SIZEOF(sResult);

PSB.FormatExt_5(sb, fmtstr, str1, str2, str3, str4, str5);

AssertEquals_Buffer(ADR(sExpected), ADR(sResult), SIZEOF(sResult));

sb.Reset();

TEST_FINISHED();
END_METHOD

METHOD T005_FormatExt_6
VAR_INPUT
	fmtstr : STRING(255);
	str1 : STRING(255);
	str2 : STRING(255);
	str3 : STRING(255);
	str4 : STRING(255);
	str5 : STRING(255);
	str6 : STRING(255);
	sExpected : STRING(500);
END_VAR
VAR_INST
	sResult : STRING(500);
	sb : PSB.StringBuilderExt;
END_VAR
TEST(concat(concat('T005_Format_6:', fmtstr), concat('-', sExpected)));

sb.pBuffer := ADR(sResult);
sb.szBuffer := SIZEOF(sResult);

PSB.FormatExt_6(sb, fmtstr, str1, str2, str3, str4, str5, str6);

AssertEquals_Buffer(ADR(sExpected), ADR(sResult), SIZEOF(sResult));
sb.Reset();
TEST_FINISHED();
END_METHOD

METHOD T006_FormatExt_7
VAR_INPUT
	fmtstr : STRING(255);
	str1 : STRING(255);
	str2 : STRING(255);
	str3 : STRING(255);
	str4 : STRING(255);
	str5 : STRING(255);
	str6 : STRING(255);
	str7 : STRING(255);
	sExpected : STRING(500);
END_VAR
VAR_INST
	sResult : STRING(500);
	sb : PSB.StringBuilderExt;
END_VAR
TEST(concat(concat('T006_Format_7:', fmtstr), concat('-', sExpected)));

sb.pBuffer := ADR(sResult);
sb.szBuffer := SIZEOF(sResult);

PSB.FormatExt_7(sb, fmtstr, str1, str2, str3, str4, str5, str6, str7);

AssertEquals_Buffer(ADR(sExpected), ADR(sResult), SIZEOF(sResult));
sb.Reset();
TEST_FINISHED();
END_METHOD

METHOD T007_FormatExt_8
VAR_INPUT
	fmtstr : STRING(255);
	str1 : STRING(255);
	str2 : STRING(255);
	str3 : STRING(255);
	str4 : STRING(255);
	str5 : STRING(255);
	str6 : STRING(255);
	str7 : STRING(255);
	str8 : STRING(255);
	sExpected : STRING(500);
END_VAR
VAR_INST
	sResult : STRING(500);
	sb : PSB.StringBuilderExt;
END_VAR
TEST(concat(concat('T007_Format_8:', fmtstr), concat('-', sExpected)));

sb.pBuffer := ADR(sResult);
sb.szBuffer := SIZEOF(sResult);

PSB.FormatExt_8(sb, fmtstr, str1, str2, str3, str4, str5, str6, str7, str8);

AssertEquals_Buffer(ADR(sExpected), ADR(sResult), SIZEOF(sResult));
sb.Reset();
TEST_FINISHED();
END_METHOD

METHOD T008_FormatExt_9
VAR_INPUT
	fmtstr : STRING(255);
	str1 : STRING(255);
	str2 : STRING(255);
	str3 : STRING(255);
	str4 : STRING(255);
	str5 : STRING(255);
	str6 : STRING(255);
	str7 : STRING(255);
	str8 : STRING(255);
	str9 : STRING(255);
	sExpected : STRING(500);
END_VAR
VAR_INST
	sResult : STRING(500);
	sb : PSB.StringBuilderExt;
END_VAR
TEST(concat(concat('T008_Format_9:', fmtstr), concat('-', sExpected)));

sb.pBuffer := ADR(sResult);
sb.szBuffer := SIZEOF(sResult);

PSB.FormatExt_9(sb, fmtstr, str1, str2, str3, str4, str5, str6, str7, str8, str9);

AssertEquals_Buffer(ADR(sExpected), ADR(sResult), SIZEOF(sResult));
sb.Reset();
TEST_FINISHED();
END_METHOD

METHOD T009_FormatExt_10
VAR_INPUT
	fmtstr : STRING(255);
	str1 : STRING(255);
	str2 : STRING(255);
	str3 : STRING(255);
	str4 : STRING(255);
	str5 : STRING(255);
	str6 : STRING(255);
	str7 : STRING(255);
	str8 : STRING(255);
	str9 : STRING(255);
	str10 : STRING(255);
	sExpected : STRING(500);
END_VAR
VAR_INST
	sResult : STRING(500);
	sb : PSB.StringBuilderExt;
END_VAR
TEST(concat(concat('T009_Format_10:', fmtstr), concat('-', sExpected)));

sb.pBuffer := ADR(sResult);
sb.szBuffer := SIZEOF(sResult);

PSB.FormatExt_10(sb, fmtstr, str1, str2, str3, str4, str5, str6, str7, str8, str9, str10);

AssertEquals_Buffer(ADR(sExpected), ADR(sResult), SIZEOF(sResult));
sb.Reset();
TEST_FINISHED();
END_METHOD

METHOD T010_FormatExt_2
VAR_INPUT
	fmtstr : STRING(255);
	i : INT;
	rl : REAL;
	sExpected : STRING(500);
END_VAR
VAR_INST
	sResult : STRING(500);
	sb : PSB.StringBuilderExt;
END_VAR
TEST(concat(concat('T010_Format_2:', fmtstr), concat('-', sExpected)));

sb.pBuffer := ADR(sResult);
sb.szBuffer := SIZEOF(sResult);

PSB.FormatExt_2(sb, fmtstr, TO_STRING(i), TO_STRING(rl));

AssertEquals_Buffer(ADR(sExpected), ADR(sResult), sizeof(sResult));
sb.Reset();
TEST_FINISHED();
END_METHOD

END_FUNCTION_BLOCK
